// TwinCAT 3 PLC project PLC_v01
// ProgramVersion: 3.1.4023.0
// libraries:
//   Tc2_Standard, * (Beckhoff Automation GmbH)
//   Tc2_System, * (Beckhoff Automation GmbH)
//   Tc3_Module, * (Beckhoff Automation GmbH)
// project tree:
//   / PlcTask.TcTTO
//   POUs/ MAIN.TcPOU
// real-time tasks:
//   TASK PlcTask: cycle T#10ms, priority 20, ADS port 350

CONFIGURATION PLC_v01
    RESOURCE PLC ON TwinCAT3
        TASK PlcTask(INTERVAL := T#10ms, PRIORITY := 20);
        PROGRAM MAIN WITH PlcTask : MAIN;
    END_RESOURCE
END_CONFIGURATION

// ---- POUs/MAIN.TcPOU
PROGRAM MAIN
VAR
	nCounter		: INT;
END_VAR


nCounter	:= nCounter + 1;

END_PROGRAM
